SUBAPPLICATION ChainOfActionsDemo (* Chain of Actions pattern demo: four TrueUntil instances chained via DONE->TRIGGER instead of one large ECC *)
  (* Standard: 61499-2; Description: Copyright (c) 2026 Meisterschulen am Ostbahnhof This program and the accompanying materials are made available under the terms of the Eclipse Public License 2.0 which is available at https://www.eclipse.org/legal/epl-2.0/ SPDX-License-Identifier: EPL-2.0 *)
  (* Version 1.0, 2026-08-31, Franz Höpfinger, Meisterschulen am Ostbahnhof, Chain of Actions design pattern (IEC 61499 primer course, Module 6, Valeriy Vyatkin, slide 66), demo application *)
  PACKAGE Meins::DesingPatterns::ChainOfActionsPattern;
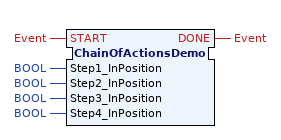
  EVENT_INPUT
    START; (* Start the chain: triggers Step1 *)
  END_EVENT
  EVENT_OUTPUT
    DONE; (* The whole chain completed (Step4 reported DONE) *)
  END_EVENT
  VAR_INPUT
    Step1_InPosition : BOOL; (* Demo: simulate Step1's actuator reaching its position *)
    Step2_InPosition : BOOL; (* Demo: simulate Step2's actuator reaching its position *)
    Step3_InPosition : BOOL; (* Demo: simulate Step3's actuator reaching its position *)
    Step4_InPosition : BOOL; (* Demo: simulate Step4's actuator reaching its position *)
  END_VAR
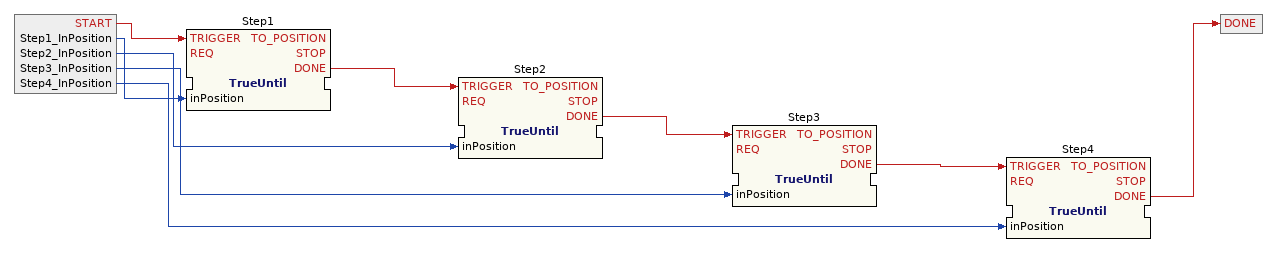
  FBS
    Step1 : Meins::DesingPatterns::ChainOfActionsPattern::TrueUntil;
    Step2 : Meins::DesingPatterns::ChainOfActionsPattern::TrueUntil;
    Step3 : Meins::DesingPatterns::ChainOfActionsPattern::TrueUntil;
    Step4 : Meins::DesingPatterns::ChainOfActionsPattern::TrueUntil;
  END_FBS
  EVENT_CONNECTIONS
    START TO Step1.TRIGGER;
    Step1.DONE TO Step2.TRIGGER;
    Step2.DONE TO Step3.TRIGGER;
    Step3.DONE TO Step4.TRIGGER;
    Step4.DONE TO DONE;
  END_CONNECTIONS
  DATA_CONNECTIONS
    Step1_InPosition TO Step1.inPosition;
    Step2_InPosition TO Step2.inPosition;
    Step3_InPosition TO Step3.inPosition;
    Step4_InPosition TO Step4.inPosition;
  END_CONNECTIONS
END_SUBAPPLICATION
